VAR_GLOBAL
	

	nullInputChannel : NullDigitalInputChannel;
	
	device1 : EL1008;
	
	myFanControlDigitalInput : AssignableDigitalInputChannel(nullInputChannel);
	
	myFanControl : TwoStateSwitch(myFanControlDigitalInput);

END_VAR

(* stored: Version 1.1.0.1, ProductVersion 3.1.4024.5
   GVL GVL_IO: Id {53f43ee1-b535-427e-9c3e-5cd19f13a68c} *)
